KUKA KRL program: FORCE.src

&ACCESS RVP1
&REL 10
&PARAM TEMPLATE = C:\KRC\Roboter\Template\FunctionVorgabe
&PARAM EDITMASK = *
DEFFCT BOOL FORCE( )

DECL INT md_int[16]
DECL REAL md_real[16]
DECL INT n
DECL INT result

FOR n=1 TO 16
md_int[n]=0
md_REAL[n]=0
ENDFOR

md_int[1]=1
md_int[2]=0
md_int[3]=0
md_real[1]=10
md_real[2]=50.0
md_real[3]=500.0
md_real[4]=0.2
md_real[5]=0.01
md_real[6]=0.01
md_real[7]=0.0

result=MD_CMD("PAPAS","DESIREDFORCEZ",md_int[],md_real[])
result=MD_CMD("PAPAS","DESIREDFORCESTART",md_int[],md_real[])

RETURN TRUE
ENDFCT
